(* CODESYS project Motors.gvl.xml

Project tree, tasks and I/O mapping:
  global variables Motors
*)

// Motors
{attribute 'qualified_only'}
VAR_GLOBAL
	AgitatorMotor: AgitatorMotor;
	BagFeedMotor: BagFeedMotor;
	BagFeedMotor_: BagFeedMotor_;
	BlowerMotor: BlowerMotor;
	HeatSealMotor: HeatSealMotor;
	IceFeedMotor: IceFeedMotor;
	KickerMotor: KickerMotor;
END_VAR
